//{{V2}}
ORGANIZATION_BLOCK OB1
TITLE= "Zyklisches Hauptprogramm"


AUTHOR:nb
FAMILY:nb
NAME:nb
VERSION:1.0


VAR_TEMP
       OB1_EV_CLASS:BYTE //Bits 0-3 = 1 (Coming event), Bits 4-7 = 1 (Event class 1)
       OB1_SCAN_1:BYTE //1 (Cold restart scan 1 of OB 1), 3 (Scan 2-n of OB 1)
       OB1_PRIORITY:BYTE //1 (Priority of 1 is lowest)
       OB1_OB_NUMBR:BYTE //1 (Organization block 1, OB1)
       OB1_RESERVED_1:BYTE //Reserved for system
       OB1_RESERVED_2:BYTE //Reserved for system
       OB1_PREV_CYCLE:INT //Cycle time of previous OB1 scan (milliseconds)
       OB1_MIN_CYCLE:INT //Minimum cycle time of OB1 (milliseconds)
       OB1_MAX_CYCLE:INT //Maximum cycle time of OB1 (milliseconds)
       OB1_DATE_TIME:DATE_AND_TIME //Date and time OB1 started
END_VAR
BEGIN

NETWORK
TITLE=Motor Schaltung
//{{k}}
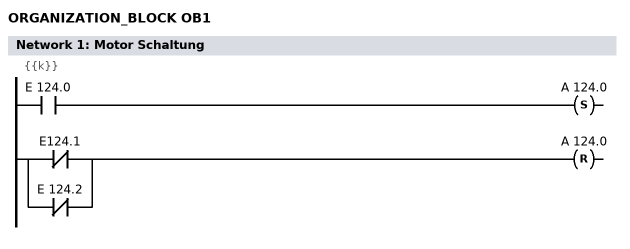

       U    E       124.0
       S    A       124.0
       U(
       ON   E124.1
       ON   E       124.2
       )
       R    A       124.0
NETWORK
TITLE=Lüfterschaltung
//{{k}}

       U    A124.0
       L    S5T#4S
       SE   T20
       NOP  0
       NOP  0
       LC   T20
       T    MW        10
       U    T20
       S    A       124.1
       UN   A       124.0
       U    A       124.1
       L    S5T#7S
       SE   T21
       NOP  0
       NOP  0
       LC   T21
       T    MW        12
       U    T21
       R    A124.1
END_ORGANIZATION_BLOCK
